FUNCTION_BLOCK TANK_MV (* Model+View for a Liquid Tank *)
  (* Standard: 61499-1 *)
  (* Version 0.2, 2001-04-23, JHC, Rockwell Automation, Moved to fb.rt.process. *)
  (* Version 0.1, 2000-06-21, JHC, Rockwell Automation, Uses LibraryElement.dtd *)
  (* Version 0.0, 2000-04-28, JHC, Rockwell Automation *)
  (* Compiler header: package fb.rt.process; import fb.rt.hmi.*; import fb.rt.math.*; *)
  (* Compiler Java IBM VisualAge 3.0 *)
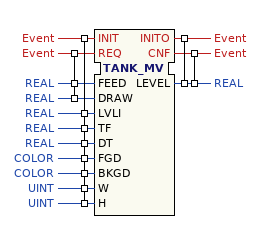
  EVENT_INPUT
    INIT WITH LVLI, TF, DT, FGD, BKGD, W, H;
    REQ WITH FEED, DRAW; (* Run a Simulation Cycle *)
  END_EVENT
  EVENT_OUTPUT
    INITO WITH LEVEL;
    CNF WITH LEVEL;
  END_EVENT
  VAR_INPUT
    FEED : REAL := 0; (* Liquid Feed Rate(0-100,Arbitrary Units) *)
    DRAW : REAL := 0; (* Liquid Drain Rate(0-100,Arbitrary Units) *)
    LVLI : REAL; (* Initial Level *)
    TF : REAL := 30; (* Filling time in seconds at(FEED-DRAW)=100 *)
    DT : REAL := 0.25; (* Integration time interval in seconds *)
    FGD : COLOR := blue; (* Foreground Color *)
    BKGD : COLOR := white; (* Background Color *)
    W : UINT; (* Bar width *)
    H : UINT; (* Bar height *)
  END_VAR
  VAR_OUTPUT
    LEVEL : REAL := 0; (* Liquid Level(0-100,Arbitrary Units) *)
  END_VAR
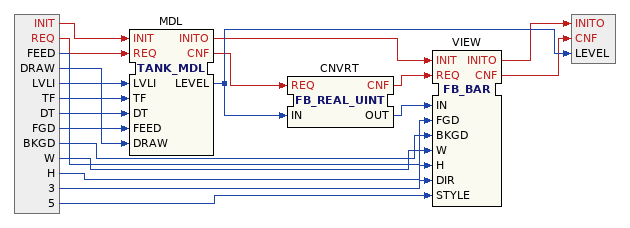
  FBS
    MDL : TANK_MDL;
    CNVRT : FB_REAL_UINT;
    VIEW : FB_BAR;
  END_FBS
  EVENT_CONNECTIONS
    INIT TO MDL.INIT;
    MDL.INITO TO VIEW.INIT;
    VIEW.INITO TO INITO;
    REQ TO MDL.REQ;
    MDL.CNF TO CNVRT.REQ;
    CNVRT.CNF TO VIEW.REQ;
    VIEW.CNF TO CNF;
  END_CONNECTIONS
  DATA_CONNECTIONS
    LVLI TO MDL.LVLI;
    TF TO MDL.TF;
    DT TO MDL.DT;
    FEED TO MDL.FEED;
    DRAW TO MDL.DRAW;
    MDL.LEVEL TO CNVRT.IN;
    MDL.LEVEL TO LEVEL;
    CNVRT.OUT TO VIEW.IN;
    FGD TO VIEW.FGD;
    BKGD TO VIEW.BKGD;
    W TO VIEW.W;
    H TO VIEW.H;
    3 TO VIEW.DIR;
    5 TO VIEW.STYLE;
  END_CONNECTIONS
END_FUNCTION_BLOCK
